(* PLC project PM, Beckhoff Automation GmbH TwinCAT PLC Control 3.5.13.21 *)
(* stored: creationDateTime 2024-07-22T16:13:01.291452, modificationDateTime 2024-07-22T16:13:01.291452 *)

{attribute 'qualified_only'}
{attribute 'strict'}
TYPE E_AnalysisIDs :
(
// Algorithms based on signal period
	Source_Period :=1,
	Frequency_Period,
	BasicValues_Period,
	PowerValues_Period,
	Harmonics_Period,
// Algorithms based on frequency domain
	Source,
	PowerValues,
	Spectrum,
	Harmonics	
) UDINT;
END_TYPE

TYPE ST_EL3773_InputSamples :
STRUCT
// Inputs from EL3773
	aUL1 : ARRAY[1..cOversamples] OF INT;
	aUL2 : ARRAY[1..cOversamples] OF INT;
	aUL3 : ARRAY[1..cOversamples] OF INT;
	aIL1 : ARRAY[1..cOversamples] OF INT;
	aIL2 : ARRAY[1..cOversamples] OF INT;
	aIL3 : ARRAY[1..cOversamples] OF INT;
END_STRUCT
END_TYPE

TYPE ST_EL3773_InputSamples_Scaled :
STRUCT
// Inputs from EL3773
	aUL1 : ARRAY[1..cOversamples] OF LREAL;
	aUL2 : ARRAY[1..cOversamples] OF LREAL;
	aUL3 : ARRAY[1..cOversamples] OF LREAL;
	aIL1 : ARRAY[1..cOversamples] OF LREAL;
	aIL2 : ARRAY[1..cOversamples] OF LREAL;
	aIL3 : ARRAY[1..cOversamples] OF LREAL;
END_STRUCT
END_TYPE

TYPE ST_Signal_HMI :
STRUCT
	aIL	 : ARRAY[1..3] OF ARRAY[1..cOversamples*cScaleHMI] OF LREAL;
	aUL	 : ARRAY[1..3] OF ARRAY[1..cOversamples*cScaleHMI] OF LREAL;
END_STRUCT
END_TYPE

FUNCTION_BLOCK FB_SystemTime
VAR_INPUT
END_VAR
VAR_OUTPUT
END_VAR
VAR
	GetLocalSystemTime 	: FB_LocalSystemTime;
	wDateW				: WORD;
END_VAR

                  GetLocalSystemTime(bEnable := TRUE);
                

PROPERTY dtDateTimeFull : DT
GET
VAR
END_VAR
                          dtDateTimeFull 	:= SYSTEMTIME_TO_DT(GetLocalSystemTime.systemTime);
                        
END_GET
END_PROPERTY

PROPERTY sDate : STRING
GET
VAR
END_VAR
                          sDate	:= MID(sDateTimeFull,10,1);
                        
END_GET
END_PROPERTY

PROPERTY sDateTime : STRING
GET
VAR
END_VAR
                          sDateTime := MID(sDateTimeFull,19,1);
                        
END_GET
END_PROPERTY

PROPERTY sDateTimeFull : STRING
GET
VAR
END_VAR
                          sDateTimeFull 	:= SYSTEMTIME_TO_STRING(GetLocalSystemTime.systemTime);
                        
END_GET
END_PROPERTY

PROPERTY sDayOfWeek : STRING
GET
VAR
END_VAR
                          wDateW	:=  GetLocalSystemTime.systemTime.wDayOfWeek;
IF wDateW = 0 THEN
	sDayOfWeek := 'Sunday';
ELSIF wDateW = 1 THEN
	sDayOfWeek := 'Monday';
ELSIF wDateW = 2 THEN
	sDayOfWeek := 'Tuesday';
ELSIF wDateW = 3 THEN
	sDayOfWeek := 'Wednesday';
ELSIF wDateW = 4 THEN
	sDayOfWeek := 'Thursday';
ELSIF wDateW = 5 THEN
	sDayOfWeek := 'Friday';
ELSIF wDateW = 6 THEN
	sDayOfWeek := 'Saturday';
END_IF
                        
END_GET
END_PROPERTY

PROPERTY sTime : STRING
GET
VAR
END_VAR
                          sTime := MID(sDateTimeFull,8,12);
                        
END_GET
END_PROPERTY

PROPERTY wDay : Word
GET
VAR
END_VAR
                          wDay :=  GetLocalSystemTime.systemTime.wDay;
                        
END_GET
END_PROPERTY

PROPERTY wHour : WORD
GET
VAR
END_VAR
                          wHour	:=	GetLocalSystemTime.systemTime.wHour;
                        
END_GET
END_PROPERTY

PROPERTY wMilliSeconds : WORD
GET
VAR
END_VAR
                          wMilliseconds	:=	GetLocalSystemTime.systemTime.wMilliseconds;
                        
END_GET
END_PROPERTY

PROPERTY wMinute : WORD
GET
VAR
END_VAR
                          wMinute	:=	GetLocalSystemTime.systemTime.wMinute;
                        
END_GET
END_PROPERTY

PROPERTY wMonth : Word
GET
VAR
END_VAR
                          wMonth	:=  GetLocalSystemTime.systemTime.wMonth;
                        
END_GET
END_PROPERTY

PROPERTY wSecond : WORD
GET
VAR
END_VAR
                          wSecond	:=	GetLocalSystemTime.systemTime.wSecond;
                        
END_GET
END_PROPERTY

PROPERTY wYear : Word
GET
VAR
END_VAR
                          wYear :=  GetLocalSystemTime.systemTime.wYear;
                        
END_GET
END_PROPERTY
END_FUNCTION_BLOCK

PROGRAM MAIN
VAR
	
	//function block
	fbScaling					: FB_PMA_Scaling_EL3773			
									:=( stInitPars	:= cScalingEL3773Pars);

	fbSource_Period				: FB_PMA_Source_3Ph 			
									:=( nOwnID		:= E_AnalysisIDs.Source_Period, 
										aDestIDs	:= [E_AnalysisIDs.Frequency_Period, 
														E_AnalysisIDs.BasicValues_Period, 
														E_AnalysisIDs.PowerValues_Period, 
														E_AnalysisIDs.Harmonics_Period],
										stInitPars	:= cSource_PeriodInitPars);
										
	fbSource					: FB_PMA_Source_3Ph				
									:=( nOwnID		:= E_AnalysisIDs.Source, 
										aDestIDs	:= [E_AnalysisIDs.PowerValues, 
														E_AnalysisIDs.Spectrum, 
														E_AnalysisIDs.Harmonics], 
										stInitPars	:= cSourceInitPars);
										
	fbFrequency					: FB_PMA_Frequency_Period_3Ph 	
									:=( nOwnID		:= E_AnalysisIDs.Frequency_Period,
										stInitPars	:= cFrequencyInitPars);
										
	fbBasicValues				: FB_PMA_BasicValues_Period_3Ph 
									:=( nOwnID		:= E_AnalysisIDs.BasicValues_Period, 
										stInitPars	:= cBasicValuesInitPars);
										
	fbPowerValues				: FB_PMA_PowerValues_Period_3Ph 		
									:=( nOwnID		:= E_AnalysisIDs.PowerValues_Period, 
										stInitPars	:= cPowerValuesPedInitPars);
										
	fbHarmonics					: FB_PMA_Harmonics_Period_3Ph 
									:=( nOwnID		:= E_AnalysisIDs.Harmonics_Period, 
										stInitPars	:= cHarmonicsPedInitPars);
	
	bResetStatistics			: BOOL;	
	
END_VAR

                  Scale();
fbSource_Period.Call(	pBuffer_UL1 		:= ADR(stEL3773_1_Scaled.aUL1),
						pBuffer_UL2 		:= ADR(stEL3773_1_Scaled.aUL2),
						pBuffer_UL3 		:= ADR(stEL3773_1_Scaled.aUL3),
						pBuffer_IL1 		:= ADR(stEL3773_1_Scaled.aIL1),
						pBuffer_IL2 		:= ADR(stEL3773_1_Scaled.aIL2),
						pBuffer_IL3 		:= ADR(stEL3773_1_Scaled.aIL3),
						nDataInSizePerCh	:= SIZEOF(stEL3773_1_Scaled.aUL1),
						nOptionPars			:= 0);
						
fbSource.Call(			pBuffer_UL1			:= ADR(stEL3773_1_Scaled.aUL1),
						 pBuffer_UL2		:= ADR(stEL3773_1_Scaled.aUL2),
						 pBuffer_UL3		:= ADR(stEL3773_1_Scaled.aUL3),
						 pBuffer_IL1		:= ADR(stEL3773_1_Scaled.aIL1),
						 pBuffer_IL2		:= ADR(stEL3773_1_Scaled.aIL2),
						 pBuffer_IL3		:= ADR(stEL3773_1_Scaled.aIL3),
						 nDataInSizePerCh	:= SIZEOF(stEL3773_1_Scaled.aUL1),
						 nOptionPars		:= 0);			
						 
fbFrequency.Call(	bResetStatistics		:= bResetStatistics);

fbBasicValues.Call(	fFreq					:= fbFrequency.aFreq[0], 
					bResetStatistics		:= bResetStatistics);
					
fbPowerValues.Call(	fFreq					:= fbFrequency.aFreq[0], 
					bResetEnergyCalc 		:= FALSE, 
					bResetStatistics		:= bResetStatistics);
					
fbHarmonics.Call(	fFreq					:= fbFrequency.aFreq[0],
					pHarmonicsRMS_UL1 		:= ADR(aHarmonicsPed[0]),
					pHarmonicsRMS_UL2 		:= ADR(aHarmonicsPed[1]),
					pHarmonicsRMS_UL3 		:= ADR(aHarmonicsPed[2]),
					pHarmonicsRMS_IL1 		:= ADR(aHarmonicsPed[3]),
					pHarmonicsRMS_IL2 		:= ADR(aHarmonicsPed[4]),
					pHarmonicsRMS_IL3 		:= ADR(aHarmonicsPed[5]),
					nHarmonicsRMSSize 		:= SIZEOF(aHarmonicsPed[0]),
					bResetStatistics		:= bResetStatistics);
						

			
                

ACTION Scale:
                      
fbScaling.Call_3Ph(	pInputBuffer_UL1	:= ADR(stEL3773_1_In.aUL1),
					pInputBuffer_UL2	:= ADR(stEL3773_1_In.aUL2),
					pInputBuffer_UL3	:= ADR(stEL3773_1_In.aUL3),
					pInputBuffer_IL1	:= ADR(stEL3773_1_In.aIL1),
					pInputBuffer_IL2	:= ADR(stEL3773_1_In.aIL2),
					pInputBuffer_IL3	:= ADR(stEL3773_1_In.aIL3),
					nInputBufferSize	:= SIZEOF(stEL3773_1_In.aUL1), 
					pOutputBuffer_UL1	:= ADR(stEL3773_1_Scaled.aUL1),
					pOutputBuffer_UL2	:= ADR(stEL3773_1_Scaled.aUL2),
					pOutputBuffer_UL3	:= ADR(stEL3773_1_Scaled.aUL3),					
					pOutputBuffer_IL1	:= ADR(stEL3773_1_Scaled.aIL1),
					pOutputBuffer_IL2	:= ADR(stEL3773_1_Scaled.aIL2),
					pOutputBuffer_IL3	:= ADR(stEL3773_1_Scaled.aIL3),
					nOutputBufferSize	:= SIZEOF(stEL3773_1_Scaled.aUL1));						
				
                    
END_ACTION
END_PROGRAM

PROGRAM MAIN_PM
VAR
	fbPowerValues				: FB_PMA_PowerValues_3Ph 	
									:=( nOwnID		:= E_AnalysisIDs.PowerValues, 
										stInitPars	:= cPowerValuesInitPars);
										
	fbSpectrum					: FB_PMA_Spectrum_3Ph		
									:=( nOwnID		:= E_AnalysisIDs.Spectrum, 
										stInitPars	:= cSpectrumInitPars);
										
	fbHarmonics					: FB_PMA_Harmonics_3Ph	 	
									:=( nOwnID		:= E_AnalysisIDs.Harmonics,
										stInitPars	:= cHarmonicsInitPars);

	bResetStatistics			: BOOL;	
	bResetEnergyCalculation		: BOOL;	
END_VAR

                  PRG_Calculate();
PRG_Database();
fbPowerValues.Call(	bResetEnergyCalc 		:= bResetEnergyCalculation,
					bResetStatistics 		:= bResetStatistics);
							
fbSpectrum.Call( pMagnitudeSpectrum_UL1 	:= ADR(aSpectrum[0]),
				pMagnitudeSpectrum_UL2 		:= ADR(aSpectrum[1]), 
				pMagnitudeSpectrum_UL3 		:= ADR(aSpectrum[2]), 
				pMagnitudeSpectrum_IL1 		:= ADR(aSpectrum[3]), 
				pMagnitudeSpectrum_IL2 		:= ADR(aSpectrum[4]), 
				pMagnitudeSpectrum_IL3 		:= ADR(aSpectrum[5]), 
				nMagnitudeSpectrumSize 		:= SIZEOF(aSpectrum[0]));

fbHarmonics.Call(	bResetStatistics 		:= bResetStatistics,
					pHarmonicsRMS_UL1 		:= ADR(aHarmonics[0]),					
					pHarmonicsRMS_UL2 		:= ADR(aHarmonics[1]),				
					pHarmonicsRMS_UL3 		:= ADR(aHarmonics[2]),
					pHarmonicsRMS_IL1 		:= ADR(aHarmonics[3]),				
					pHarmonicsRMS_IL2 		:= ADR(aHarmonics[4]),
					pHarmonicsRMS_IL3 		:= ADR(aHarmonics[5]),
					nHarmonicsRMSSize 		:= SIZEOF(aHarmonics[0]));
							
                
END_PROGRAM

PROGRAM PRG_Calculate
VAR
		state, m, n, i, j, k, t		: UDINT := 1;
END_VAR

                  //========== Frequency calculate ========//
fSampleRate							  := cOversamples * (1000.0 / fSampleTaskCycleTime);
fResolution 						  := fSampleRate / cFFTLength;	

//========== Create array for HMI ========//
IF timeArray[cScaleHMI*cOversamples] <> cScaleHMI*cOversamples THEN
	FOR n := 1 TO cScaleHMI*cOversamples DO timeArray[n] := n;	END_FOR
	FOR t := 1 TO cFFTResult 			 DO freqArray[t] := (t-1)*fResolution;	END_FOR
END_IF

IF m < cScaleHMI THEN
	FOR j := 1 TO cOversamples DO //fill first data to HMI array
		signal_UI.aIL[1][(m-1)*10+j]  := stEL3773_1_Scaled.aIL1[j];
		signal_UI.aIL[2][(m-1)*10+j]  := stEL3773_1_Scaled.aIL2[j];
		signal_UI.aIL[3][(m-1)*10+j]  := stEL3773_1_Scaled.aIL3[j];
		signal_UI.aUL[1][(m-1)*10+j]  := stEL3773_1_Scaled.aUL1[j];
		signal_UI.aUL[2][(m-1)*10+j]  := stEL3773_1_Scaled.aUL2[j];
		signal_UI.aUL[3][(m-1)*10+j]  := stEL3773_1_Scaled.aUL3[j];		
	END_FOR
	m := m + 1;
ELSE
	m := cScaleHMI;
	FOR i := 1 TO cScaleHMI-1 DO
		FOR j := 1 TO cOversamples DO //move data to 1st slot empty
			signal_UI.aIL[1][(i-1)*10+j]	:= signal_UI.aIL[1][(i)*10+j];
			signal_UI.aIL[2][(i-1)*10+j]	:= signal_UI.aIL[2][(i)*10+j];
			signal_UI.aIL[3][(i-1)*10+j]	:= signal_UI.aIL[3][(i)*10+j];	
			signal_UI.aUL[1][(i-1)*10+j]	:= signal_UI.aUL[1][(i)*10+j];
			signal_UI.aUL[2][(i-1)*10+j]	:= signal_UI.aUL[2][(i)*10+j];
			signal_UI.aUL[3][(i-1)*10+j]	:= signal_UI.aUL[3][(i)*10+j];				
		END_FOR
	END_FOR
	FOR k := 1 TO cOversamples DO //newest data in the 1st slot
		signal_UI.aIL[1][(m-1)*10+k]  := stEL3773_1_Scaled.aIL1[k];
		signal_UI.aIL[2][(m-1)*10+k]  := stEL3773_1_Scaled.aIL2[k];
		signal_UI.aIL[3][(m-1)*10+k]  := stEL3773_1_Scaled.aIL3[k];
		signal_UI.aUL[1][(m-1)*10+k]  := stEL3773_1_Scaled.aUL1[k];
		signal_UI.aUL[2][(m-1)*10+k]  := stEL3773_1_Scaled.aUL2[k];
		signal_UI.aUL[3][(m-1)*10+k]  := stEL3773_1_Scaled.aUL3[k];		
	END_FOR	
END_IF	
                
END_PROGRAM

PROGRAM PRG_Database
VAR
	fbSystemTime			: FB_SystemTime;
	bSaveData				: BOOL;
	bLoadData				: BOOL;
	nStateSave, nStateLoad	: INT;
	tTimer1, tTimer2		: TON;
	bTest					: BOOL;
	nStateADS				: INT;
END_VAR

                  fbSystemTime();
sCurrentTime	:= fbSystemTime.sTime;
nCurrentSec		:= fbSystemTime.wSecond;
CASE nStateSave OF
	0:
		tTimer1(IN := FALSE);
		IF nCurrentSec = 70 OR sCurrentTime = '06:00:00' OR sCurrentTime = '14:00:00' OR sCurrentTime = '22:00:00' THEN
			nStateSave			:= 1;
		END_IF
	1:
		aFFTU1						:= aSpectrum[0];
		aFFTU2						:= aSpectrum[1];
		aFFTU3						:= aSpectrum[2];
		
		aFFTI1						:= aSpectrum[3];
		aFFTI2						:= aSpectrum[4];
		aFFTI3						:= aSpectrum[5];
		
		RMSI1						:= MAIN.fbBasicValues.aRMS_I[0]/2.44;
		RMSI2						:= MAIN.fbBasicValues.aRMS_I[1]/2.44;
		RMSI3						:= MAIN.fbBasicValues.aRMS_I[2]/2.44;
		
		RMSU1						:= MAIN.fbBasicValues.aRMS_U[0];
		RMSU2						:= MAIN.fbBasicValues.aRMS_U[1];
		RMSU3						:= MAIN.fbBasicValues.aRMS_U[2];		
		
		Frequency					:= LREAL_TO_REAL(MAIN.fbFrequency.aFreq[0]);
		
		bAddData					:= TRUE;
		nStateSave					:= 2;
	2:
		IF NOT bAddData THEN
			tTimer1(IN := TRUE,PT := T#2S);
			IF tTimer1.Q THEN
				nStateSave			:= 0;		
			END_IF	
		END_IF
			
		
END_CASE

CASE nStateADS OF
	0:
		IF bCheckADS THEN
			nStateADS := 1;
		ELSE
			tTimer2(IN := TRUE,PT := T#5S);
			IF tTimer2.Q THEN
				nStateADS := 2;
			END_IF
		END_IF
		
	1:
		bCheckADS := FALSE;
		bError	:= FALSE;
		tTimer2(IN := FALSE);
		nStateADS := 0;
	2:
		bError := TRUE;
		tTimer2(IN := FALSE);
		IF bCheckADS THEN
			nStateADS := 0;
		END_IF
END_CASE
                
END_PROGRAM

CONFIGURATION Application
  RESOURCE PM ON PLC
(* global variable list GVL *)
VAR_GLOBAL CONSTANT
	cOversamples				: UDINT 					:= 10;					// number of oversamples
	cSamplerate					: UDINT 					:= 1000 * cOversamples;	// samplerate
	cFFTLength					: UDINT 					:= 4096;				// length of fft
	cWindowLength				: UDINT 					:= 3200;				// internal buffer size with 50% overlapping
	cBufferLength				: UDINT 					:= cWindowLength/2;		// buffer size
	cHarmonicBands				: UDINT 					:= 20;					// number of harmonics
	cFreqMode					: LREAL 					:= 50.0;				// base frequency	
	cFFTResult					: UDINT						:= cFFTLength/2 +1;
	cScaleHMI					: UDINT						:= 250;
	//FB_Scaling signal from IO s
	cScalingEL3773Pars			: ST_PMA_Scaling_EL3773_InitPars 	 	
									:=( nOversamples 		:= cOversamples, 
										fOffsetVoltage 		:= 0, 
										fGainVoltage 		:= 1, 
										fOffsetCurrent 		:= 0, 
										fGainCurrent 		:= 1, 
										fFactorCurrentTransformer := 100); //In/Out value of CT
	
	//FB_Source for period
	cSource_PeriodInitPars		: ST_PMA_Source_InitPars 		 		
									:=( nBufferLength 		:= cOversamples);	
	
	//FB_Source freq domain								
	cSourceInitPars				: ST_PMA_Source_InitPars 				
									:=( nBufferLength 		:= cBufferLength);
		
	//FB_Frequence - period							
	cFrequencyInitPars			: ST_PMA_Frequency_Period_InitPars 		
									:=( nBufferLength 		:= cOversamples, 
										fSampleRate 		:= cSamplerate, 
										fMinFreq 			:= 10, 
										fMaxFreq 			:= 70, 
										nPeriods 			:= 10, 
										nFilterOrder 		:= 2, 
										fCutoff 			:= 70, 
										eInputSelect 		:= E_PMA_InputSelect.Current, 
										fMinInput 			:= 0);
	
	//Basic value in time domain									
	cBasicValuesInitPars		: ST_PMA_BasicValues_Period_InitPars 	
									:=( nBufferLength 		:= cOversamples, 
										fSampleRate 		:= cSamplerate, 
										fMinInputCurrent 	:= 0.0,
										nPeriods         	:= 20 );
	
	//Power value in period									
	cPowerValuesPedInitPars		: ST_PMA_PowerValues_Period_InitPars 	
									:=( nBufferLength 		:= cOversamples, 
										fSampleRate 		:= cSamplerate, 
										fMinInputCurrent 	:= 0.0,
										nPeriods			:= 10);
		
	//Harmonics in period								
	cHarmonicsPedInitPars		: ST_PMA_Harmonics_Period_InitPars		
									:=( nBufferLength 		:= cOversamples, 
										fSampleRate 		:= cSamplerate, 
										nNumHarmonics 		:= cHarmonicBands, 
										nPeriods 			:= 10, 
										bTransformToPercent := TRUE);
											
	//Power value in freq domain
	cPowerValuesInitPars		: ST_PMA_PowerValues_InitPars
									:=( uTimeLagCurrentTransformer := (aTimeLag := [0.0, 0.0, 0.0]),
										fSampleRate 		:= cSamplerate,			// in Hz 
										fBaseFreq 			:= cFreqMode,			// in Hz
										nFFT_Length 		:= cFFTLength,
										nWindowLength 		:= cWindowLength,
										nNumBands 			:= 20,
										fBandwidth 			:= 20.0,
										fMinInputCurrent	:= 0.0,
										eWindowType 		:= E_PMA_WindowType.HannWindow);
										
	// FB_PMA_Spectrum in freq domain
	cSpectrumInitPars			: ST_PMA_Spectrum_InitPars
									:=(	nFFT_Length 		:= cFFTLength,
										nWindowLength 		:= cWindowLength, 
										fSampleRate 		:= cSamplerate,			// in Hz
										bTransformToDecibel := FALSE,
										eWindowType 		:= E_PMA_WindowType.HannWindow,
										eScalingType 		:= E_PMA_ScalingType.RMS);	
										
	// FB_PMA_Harmonics	in freq domain								
	cHarmonicsInitPars			: ST_PMA_Harmonics_InitPars
									:=(	nFFT_Length 		:= cFFTLength,
										nWindowLength 		:= cWindowLength,
										fSampleRate 		:= cSamplerate,			// in Hz
										nNumBands 			:= cHarmonicBands,
										fBaseFreq 			:= cFreqMode,			// in Hz
										fBandwidth 			:= 20.0,
										eWindowType 		:= E_PMA_WindowType.HannWindow,	
										bTransformToDecibel := FALSE,
										bTransformToPercent := FALSE);	
END_VAR

VAR_GLOBAL
	stEL3773_1_In 			AT%I* 	: ST_EL3773_InputSamples;
	stEL3773_1_Scaled				: ST_EL3773_InputSamples_Scaled;	
	signal_UI						: ST_Signal_HMI;
	signal_UI_Zeros					: ST_Signal_HMI;
	

	fSampleTaskCycleTime			: LREAL := 1; 	// ms
	fSampleRate						: LREAL; 		// Hz  ( sample rate = oversampling factor / cycle time )
	fResolution						: LREAL; 		// Hz/Idx		
	sendArray						: BOOL;
	timeArray						: ARRAY[1..cOversamples*cScaleHMI] OF UDINT;
	freqArray						: ARRAY[1..cFFTResult] OF LREAL;
	aHarmonicsPed 					: ARRAY[0..5] OF ARRAY [0..cHarmonicBands-1] OF LREAL; 
	
	aSpectrum						: ARRAY[0..5] OF ARRAY [0..cFFTLength/2] OF LREAL;		// dims: [UL1..UL3 + IL1..IL3][FFTLength/2 + 1]
	aHarmonics						: ARRAY[0..5] OF ARRAY [0..cHarmonicBands-1] OF LREAL;	// dims: [UL1..UL3 + IL1..IL3][NumBands]

	nCurrentDate					: WORD;
	sCurrentTime					: STRING;
	nCurrentHour					: WORD;
	nCurrentSec						: WORD;		
	wFreq		AT %Q*	: WORD;
END_VAR

VAR_GLOBAL PERSISTENT
	alarmCurrent					: ARRAY [1..2] OF ARRAY [1..3] OF LREAL; //1 : alram, 2 : warning
	alarmVoltage					: ARRAY [1..2] OF ARRAY [1..3] OF LREAL;	
	
END_VAR
(* global variable list GVL_ADS *)
VAR_GLOBAL
	aFFTI1 					: ARRAY[1..cFFTResult] OF LREAL;
	aFFTI2					: ARRAY[1..cFFTResult] OF LREAL;
	aFFTI3					: ARRAY[1..cFFTResult] OF LREAL;
	RMSI1					: LREAL;
	RMSI2					: LREAL;
	RMSI3					: LREAL;
	Frequency				: REAL;
	
	aFFTU1 					: ARRAY[1..cFFTResult] OF LREAL;
	aFFTU2					: ARRAY[1..cFFTResult] OF LREAL;
	aFFTU3					: ARRAY[1..cFFTResult] OF LREAL;
	RMSU1					: LREAL;
	RMSU2					: LREAL;
	RMSU3					: LREAL;	
	//bAdd
	bAddData				: BOOL;
	bCheckADS				: BOOL;
	bError					: BOOL;
END_VAR
    TASK PlcTask(INTERVAL := T#0ms, PRIORITY := 6);
    TASK PlcTaskPM(INTERVAL := T#0ms, PRIORITY := 16);
    TASK TaskCalc(INTERVAL := T#0ms, PRIORITY := 8);
    PROGRAM MAIN WITH PlcTask : MAIN;
    PROGRAM MAIN_PM WITH PlcTaskPM : MAIN_PM;
    PROGRAM PRG_Calculate WITH TaskCalc : PRG_Calculate;
  END_RESOURCE
END_CONFIGURATION
